FUNCTION_BLOCK ASSEMBLE_AW_FROM_AQ (* this Function combines the 8 AQ (QUARTER) adapters to a AW (WORD) *)
  (* Standard: 61499-2; Description: Copyright (c) 2026 Meisterschulen am Ostbahnhof SPDX-License-Identifier: EPL-2.0 *)
  (* Version 1.0, 2026-05-16, Franz Höpfinger, Meisterschulen am Ostbahnhof, initial API and implementation and/or initial documentation *)
  PACKAGE adapter::assembling;
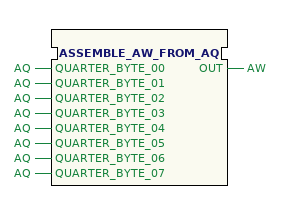
  SOCKETS
    QUARTER_BYTE_00 : adapter::types::unidirectional::AQ; (* Quarter 0 *)
    QUARTER_BYTE_01 : adapter::types::unidirectional::AQ; (* Quarter 1 *)
    QUARTER_BYTE_02 : adapter::types::unidirectional::AQ; (* Quarter 2 *)
    QUARTER_BYTE_03 : adapter::types::unidirectional::AQ; (* Quarter 3 *)
    QUARTER_BYTE_04 : adapter::types::unidirectional::AQ; (* Quarter 4 *)
    QUARTER_BYTE_05 : adapter::types::unidirectional::AQ; (* Quarter 5 *)
    QUARTER_BYTE_06 : adapter::types::unidirectional::AQ; (* Quarter 6 *)
    QUARTER_BYTE_07 : adapter::types::unidirectional::AQ; (* Quarter 7 *)
  END_SOCKETS
  PLUGS
    OUT : adapter::types::unidirectional::AW; (* WORD Output *)
  END_PLUGS
END_FUNCTION_BLOCK
